(* IEC 61131-3 sources: eCockpitGit/test_project/src/%F%00 Library/%F%Common Functions/%F%Swap Values, 13 files *)

(* ---- %POU%FU_bSwap.st ---- *)
//This function swaps two values
// +-----------+----------+----------+-----------------------------------------------------------------------------------------------------------------------+
// |**Version**|**Author**| **Date** |**Changes**                                                                                                            |
// +-----------+----------+----------+-----------------------------------------------------------------------------------------------------------------------+
// | 1         | NSN      | 13-06-18 | Updated to new guidelines                                                                                             |
// +-----------+----------+----------+-----------------------------------------------------------------------------------------------------------------------+
FUNCTION FU_bSwap : BOOL
VAR_IN_OUT
	uiA		:BYTE;		//Value a to be swapped with b
	uiB		:BYTE;		//Value b to be swapped with a
END_VAR
VAR
	C		:BYTE;		//Holding variable
END_VAR
(*%!%__DELIMITER__%!%*)
C		:=		uiA;
uiA		:=		uiB;
uiB		:=		C;

(* ---- %POU%FU_diSwap.st ---- *)
//This function swaps two values
// +-----------+----------+----------+-----------------------------------------------------------------------------------------------------------------------+
// |**Version**|**Author**| **Date** |**Changes**                                                                                                            |
// +-----------+----------+----------+-----------------------------------------------------------------------------------------------------------------------+
// | 1         | NSN      | 13-06-18 | Updated to new guidelines                                                                                             |
// +-----------+----------+----------+-----------------------------------------------------------------------------------------------------------------------+
FUNCTION FU_diSwap : BOOL
VAR_IN_OUT
	uiA		:DINT;		//Value a to be swapped with b
	uiB		:DINT;		//Value b to be swapped with a
END_VAR
VAR
	C		:DINT;		//Holding variable
END_VAR
(*%!%__DELIMITER__%!%*)
C		:=		uiA;
uiA		:=		uiB;
uiB		:=		C;

(* ---- %POU%FU_dwSwap.st ---- *)
//This function swaps two values
// +-----------+----------+----------+-----------------------------------------------------------------------------------------------------------------------+
// |**Version**|**Author**| **Date** |**Changes**                                                                                                            |
// +-----------+----------+----------+-----------------------------------------------------------------------------------------------------------------------+
// | 1         | NSN      | 13-06-18 | Updated to new guidelines                                                                                             |
// +-----------+----------+----------+-----------------------------------------------------------------------------------------------------------------------+
FUNCTION FU_dwSwap : BOOL
VAR_IN_OUT
	uiA		:DWORD;		//Value a to be swapped with b
	uiB		:DWORD;		//Value b to be swapped with a
END_VAR
VAR
	C		:DWORD;		//Holding variable
END_VAR
(*%!%__DELIMITER__%!%*)
C		:=		uiA;
uiA		:=		uiB;
uiB		:=		C;

(* ---- %POU%FU_iSwap.st ---- *)
//This function swaps two values
// +-----------+----------+----------+-----------------------------------------------------------------------------------------------------------------------+
// |**Version**|**Author**| **Date** |**Changes**                                                                                                            |
// +-----------+----------+----------+-----------------------------------------------------------------------------------------------------------------------+
// | 1         | NSN      | 13-06-18 | Updated to new guidelines                                                                                             |
// +-----------+----------+----------+-----------------------------------------------------------------------------------------------------------------------+
FUNCTION FU_iSwap : BOOL
VAR_IN_OUT
	uiA		:INT;		//Value a to be swapped with b
	uiB		:INT;		//Value b to be swapped with a
END_VAR
VAR
	C		:INT;		//Holding variable
END_VAR
(*%!%__DELIMITER__%!%*)
C		:=		uiA;
uiA		:=		uiB;
uiB		:=		C;

(* ---- %POU%FU_rSwap.st ---- *)
//This function swaps two values
// +-----------+----------+----------+-----------------------------------------------------------------------------------------------------------------------+
// |**Version**|**Author**| **Date** |**Changes**                                                                                                            |
// +-----------+----------+----------+-----------------------------------------------------------------------------------------------------------------------+
// | 1         | NSN      | 13-06-18 | Updated to new guidelines                                                                                             |
// +-----------+----------+----------+-----------------------------------------------------------------------------------------------------------------------+
FUNCTION FU_rSwap : BOOL
VAR_IN_OUT
	uiA		:REAL;		//Value a to be swapped with b
	uiB		:REAL;		//Value b to be swapped with a
END_VAR
VAR
	C		:REAL;		//Holding variable
END_VAR
(*%!%__DELIMITER__%!%*)
C		:=		uiA;
uiA		:=		uiB;
uiB		:=		C;

(* ---- %POU%FU_siSwap.st ---- *)
//This function swaps two values
// +-----------+----------+----------+-----------------------------------------------------------------------------------------------------------------------+
// |**Version**|**Author**| **Date** |**Changes**                                                                                                            |
// +-----------+----------+----------+-----------------------------------------------------------------------------------------------------------------------+
// | 1         | NSN      | 13-06-18 | Updated to new guidelines                                                                                             |
// +-----------+----------+----------+-----------------------------------------------------------------------------------------------------------------------+
FUNCTION FU_siSwap : BOOL
VAR_IN_OUT
	uiA		:SINT;		//Value a to be swapped with b
	uiB		:SINT;		//Value b to be swapped with a
END_VAR
VAR
	C		:SINT;		//Holding variable
END_VAR
(*%!%__DELIMITER__%!%*)
C		:=		uiA;
uiA		:=		uiB;
uiB		:=		C;

(* ---- %POU%FU_Swap.st ---- *)
//This function swaps two values
// +-----------+----------+----------+-----------------------------------------------------------------------------------------------------------------------+
// |**Version**|**Author**| **Date** |**Changes**                                                                                                            |
// +-----------+----------+----------+-----------------------------------------------------------------------------------------------------------------------+
// | 1         | NSN      | 21-03-19 | Creation                                                                                                              |
// +-----------+----------+----------+-----------------------------------------------------------------------------------------------------------------------+
FUNCTION FU_Swap : BOOL
VAR_INPUT
	A		:ANY;		//Value a to be swapped with b, this is the
	B		:ANY;		//Value b to be swapped with a
END_VAR
VAR
	C		:BYTE;		//Holding variable
END_VAR
(*%!%__DELIMITER__%!%*)
WHILE A.diSize > 0 DO
	C			:=		A.pValue^;
	A.pValue^	:=		B.pValue^;
	B.pValue^	:=		C;
	A.diSize	:=		A.diSize - 1;
	A.pValue	:=		A.pValue + 1;
	B.pValue	:=		B.pValue + 1;
END_WHILE

(* ---- %POU%FU_SwapAT.st ---- *)
//This function swaps two values
// +-----------+----------+----------+-----------------------------------------------------------------------------------------------------------------------+
// |**Version**|**Author**| **Date** |**Changes**                                                                                                            |
// +-----------+----------+----------+-----------------------------------------------------------------------------------------------------------------------+
// | 1         | NSN      | 21-03-19 | Creation                                                                                                              |
// +-----------+----------+----------+-----------------------------------------------------------------------------------------------------------------------+
FUNCTION FU_SwapAT : BOOL
VAR_INPUT
	A		:POINTER TO BYTE;		//Value a to be swapped with b,
	B		:POINTER TO BYTE;		//Value b to be swapped with a
	Size	:DINT;
END_VAR
VAR
	C		:BYTE;					//Holding variable
END_VAR
(*%!%__DELIMITER__%!%*)
WHILE Size > 0 DO
	C		:=		A^;
	A^		:=		B^;
	B^		:=		C;
	Size	:=		Size - 1;
	A		:=		A + 1;
	B		:=		B + 1;
END_WHILE

(* ---- %POU%FU_udiSwap.st ---- *)
//This function swaps two values
// +-----------+----------+----------+-----------------------------------------------------------------------------------------------------------------------+
// |**Version**|**Author**| **Date** |**Changes**                                                                                                            |
// +-----------+----------+----------+-----------------------------------------------------------------------------------------------------------------------+
// | 1         | NSN      | 13-06-18 | Updated to new guidelines                                                                                             |
// +-----------+----------+----------+-----------------------------------------------------------------------------------------------------------------------+
FUNCTION FU_udiSwap : BOOL
VAR_IN_OUT
	uiA		:UDINT;		//Value a to be swapped with b
	uiB		:UDINT;		//Value b to be swapped with a
END_VAR
VAR
	C		:UDINT;		//Holding variable
END_VAR
(*%!%__DELIMITER__%!%*)
C		:=		uiA;
uiA		:=		uiB;
uiB		:=		C;

(* ---- %POU%FU_uiSwap.st ---- *)
//This function swaps two values
// +-----------+----------+----------+-----------------------------------------------------------------------------------------------------------------------+
// |**Version**|**Author**| **Date** |**Changes**                                                                                                            |
// +-----------+----------+----------+-----------------------------------------------------------------------------------------------------------------------+
// | 1         | NSN      | 13-06-18 | Updated to new guidelines                                                                                             |
// +-----------+----------+----------+-----------------------------------------------------------------------------------------------------------------------+
FUNCTION FU_uiSwap : BOOL
VAR_IN_OUT
	uiA		:UINT;		//Value a to be swapped with b
	uiB		:UINT;		//Value b to be swapped with a
END_VAR
VAR
	C		:UINT;		//Holding variable
END_VAR
(*%!%__DELIMITER__%!%*)
C		:=		uiA;
uiA		:=		uiB;
uiB		:=		C;

(* ---- %POU%FU_usiSwap.st ---- *)
//This function swaps two values
// +-----------+----------+----------+-----------------------------------------------------------------------------------------------------------------------+
// |**Version**|**Author**| **Date** |**Changes**                                                                                                            |
// +-----------+----------+----------+-----------------------------------------------------------------------------------------------------------------------+
// | 1         | NSN      | 13-06-18 | Updated to new guidelines                                                                                             |
// +-----------+----------+----------+-----------------------------------------------------------------------------------------------------------------------+
FUNCTION FU_usiSwap : BOOL
VAR_IN_OUT
	uiA		:USINT;		//Value a to be swapped with b
	uiB		:USINT;		//Value b to be swapped with a
END_VAR
VAR
	C		:USINT;		//Holding variable
END_VAR
(*%!%__DELIMITER__%!%*)
C		:=		uiA;
uiA		:=		uiB;
uiB		:=		C;

(* ---- %POU%FU_wSwap.st ---- *)
//This function swaps two values
// +-----------+----------+----------+-----------------------------------------------------------------------------------------------------------------------+
// |**Version**|**Author**| **Date** |**Changes**                                                                                                            |
// +-----------+----------+----------+-----------------------------------------------------------------------------------------------------------------------+
// | 1         | NSN      | 13-06-18 | Updated to new guidelines                                                                                             |
// +-----------+----------+----------+-----------------------------------------------------------------------------------------------------------------------+
FUNCTION FU_wSwap : BOOL
VAR_IN_OUT
	uiA		:WORD;		//Value a to be swapped with b
	uiB		:WORD;		//Value b to be swapped with a
END_VAR
VAR
	C		:WORD;		//Holding variable
END_VAR
(*%!%__DELIMITER__%!%*)
C		:=		uiA;
uiA		:=		uiB;
uiB		:=		C;

(* ---- %POU%FU_xSwap.st ---- *)
//This function swaps two values
// +-----------+----------+----------+-----------------------------------------------------------------------------------------------------------------------+
// |**Version**|**Author**| **Date** |**Changes**                                                                                                            |
// +-----------+----------+----------+-----------------------------------------------------------------------------------------------------------------------+
// | 1         | NSN      | 13-06-18 | Updated to new guidelines                                                                                             |
// +-----------+----------+----------+-----------------------------------------------------------------------------------------------------------------------+
FUNCTION FU_xSwap : BOOL
VAR_IN_OUT
	uiA		:BOOL;		//Value a to be swapped with b
	uiB		:BOOL;		//Value b to be swapped with a
END_VAR
VAR
	C		:BOOL;		//Holding variable
END_VAR
(*%!%__DELIMITER__%!%*)
C		:=		uiA;
uiA		:=		uiB;
uiB		:=		C;
